{attribute 'GeneratedUsingTerminal: KL9900-0063'}
{attribute addProperty BoxType "KL9900-0063"}
{attribute addProperty Description ""}
{attribute addProperty Physics ""}
{attribute addProperty Id "Channel_1AT %Q*Channel_6CC0E2260"}
{attribute addProperty CRC "1326296452"}
{attribute addProperty Size "0"}
TYPE KL_4F0DAD84 :
STRUCT
	{attribute addProperty Name "Channel_1"}
	Channel_1 : Channel_6CC0E226;
END_STRUCT
END_TYPE

(* stored: Version 1.2.0.0, ProductVersion 3.1.4024.11
   DUT KL_4F0DAD84: Id {459758b9-b4fb-49ad-bc4d-4ecfe50c0608} *)
